// TIA Portal V17 export
// export: Created 2022-06-19T07:22:13.3877944Z, ExportSetting None, DisplayName Totally Integrated Automation Portal, DisplayVersion V17, DisplayName TIA Portal Openness, DisplayVersion V17, DisplayName TIA Portal Teamcenter Gateway, DisplayVersion V17, DisplayName TIA Portal Version Control Interface, DisplayVersion V17, DisplayName TIA Portal Test Suite Advanced, DisplayVersion V17, DisplayName SINAMICS Startdrive Advanced, DisplayVersion V17, DisplayName SINAMICS DCC, DisplayVersion V17, DisplayName SINAMICS Startdrive G130, G150, S120, S150, SINAMICS MV, S210, DisplayVersion V17, DisplayName SINAMICS Startdrive G110M, G120, G120C, G120D, G120P, G115D, DisplayVersion V17, DisplayName STEP 7 Professional, DisplayVersion V17, DisplayName SIMATIC Energy Suite, DisplayVersion V17, DisplayName STEP 7 CFC, DisplayVersion V17, DisplayName STEP 7 Safety, DisplayVersion V17, DisplayName WinCC Advanced / Unified PC, DisplayVersion V17, DisplayName SIMATIC Visualization Architect, DisplayVersion V17
DATA_BLOCK "InstanceDB_UDT"   // DB8
TITLE = TestTitle
{ S7_Optimized_Access := 'TRUE' }
AUTHOR : AV
FAMILY : Fam
NAME : eeee
VERSION : 0.11
// Comment
// stored: InstanceOfName Lib_UDT_Motor_DS_RotSens, InstanceOfType UDT
"Lib_UDT_Motor_DS_RotSens"
   // VAR RETAIN
   //    ID { S7_SetPoint := 'True'} : Int;
   //    CLSID { S7_SetPoint := 'True'} : Int;
   //    Mode { ExternalAccessible := 'False'; ExternalVisible := 'False'; ExternalWritable := 'False'} : "UDT_Mode";
   //    State { ExternalAccessible := 'False'; ExternalVisible := 'False'; ExternalWritable := 'False'} : "_Motor_DS_RotSens_StateBits";
   //    Alarm { ExternalAccessible := 'False'; ExternalVisible := 'False'; ExternalWritable := 'False'} : "_Motor_DS_RotSens_AlarmBits";
   //    CMD : Int;
   //    Config { S7_SetPoint := 'True'} : "_Motor_DS_RotSens_Config";
   //    Counters { ExternalWritable := 'False'; S7_SetPoint := 'True'} : "_Motor_DS_RotSens_Counters";
   //    Status { ExternalWritable := 'False'} : "_Motor_DS_RotSens_StateHMI";
   // END_VAR
BEGIN
END_DATA_BLOCK
